{attribute 'qualified_only'}
VAR_GLOBAL
	iNumerRamki								: INT := 0;
	
END_VAR

(* stored: Version 1.1.0.1, ProductVersion 3.1.4024.11
   GVL GVL_Wizualizacja: Id {2f53dabf-697c-41d5-86fa-88d505a144ed} *)
